SUBAPPLICATION Uebung_006a3_sub (* Subapplication Type *)
  (* Standard: 61499-2; Description: Copyright (c) 2025 Meisterschulen am Ostbahnhof This program and the accompanying materials are made available under the terms of the Eclipse Public License 2.0 which is available at https://www.eclipse.org/legal/epl-2.0/ SPDX-License-Identifier: EPL-2.0 *)
  (* Version 1.0, 2025-05-06, Franz Höpfinger, Meisterschulen am Ostbahnhof *)
  PACKAGE Uebungen;
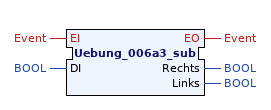
  EVENT_INPUT
    EI;
  END_EVENT
  EVENT_OUTPUT
    EO;
  END_EVENT
  VAR_INPUT
    DI : BOOL;
  END_VAR
  VAR_OUTPUT
    Rechts : BOOL;
    Links : BOOL;
  END_VAR
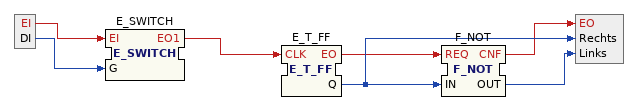
  FBS
    E_T_FF : iec61499::events::E_T_FF;
    E_SWITCH : iec61499::events::E_SWITCH;
    F_NOT : iec61131::bitwiseOperators::F_NOT;
  END_FBS
  EVENT_CONNECTIONS
    E_T_FF.EO TO F_NOT.REQ;
    EI TO E_SWITCH.EI;
    F_NOT.CNF TO EO;
    E_SWITCH.EO1 TO E_T_FF.CLK;
  END_CONNECTIONS
  DATA_CONNECTIONS
    E_T_FF.Q TO F_NOT.IN;
    E_T_FF.Q TO Rechts;
    DI TO E_SWITCH.G;
    F_NOT.OUT TO Links;
  END_CONNECTIONS
END_SUBAPPLICATION
